FUNCTION_BLOCK StandardSection (* Composite Function Block Type *)
  (* Standard: 61499-2 *)
  (* Version 0.0, 9/24/2018, dmidro, nxtControl GmbH, template *)
  PACKAGE Main;
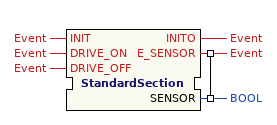
  EVENT_INPUT
    INIT; (* Initialization Request *)
    DRIVE_ON; (* Set Event *)
    DRIVE_OFF; (* Reset Event *)
  END_EVENT
  EVENT_OUTPUT
    INITO; (* Initialization Confirm *)
    E_SENSOR WITH SENSOR; (* Event Output *)
  END_EVENT
  VAR_OUTPUT
    SENSOR : BOOL; (* Current value(i) in the named variable array element *)
  END_VAR
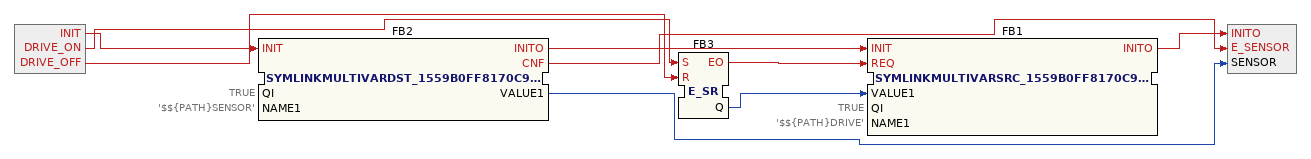
  FBS
    FB1 : SYMLINKMULTIVARSRC_1559B0FF8170C9BA0(QI := TRUE, NAME1 := '$${PATH}DRIVE'); {SET_ATTRIBUTE(Configuration.GenericFBType.InterfaceParams, Runtime.System#I:=1;VALUE${I$}:BOOL)}
    FB2 : SYMLINKMULTIVARDST_1559B0FF8170C9BA0(QI := TRUE, NAME1 := '$${PATH}SENSOR'); {SET_ATTRIBUTE(Configuration.GenericFBType.InterfaceParams, Runtime.System#I:=1;VALUE${I$}:BOOL)}
    FB3 : E_SR;
  END_FBS
  EVENT_CONNECTIONS
    INIT TO FB2.INIT;
    FB1.INITO TO INITO;
    FB2.INITO TO FB1.INIT;
    DRIVE_ON TO FB3.S;
    DRIVE_OFF TO FB3.R;
    FB3.EO TO FB1.REQ;
    FB2.CNF TO E_SENSOR;
  END_CONNECTIONS
  DATA_CONNECTIONS
    FB3.Q TO FB1.VALUE1;
    FB2.VALUE1 TO SENSOR;
  END_CONNECTIONS
END_FUNCTION_BLOCK
